// TIA Portal V19 export
DATA_BLOCK "PnPnLeftX2P1PNPortStatus_DB"   // DB11
// stored: InstanceOfName PN Port Status, InstanceOfType FB
"PN Port Status"
   // VAR_INPUT
   //    HW_ID : HW_IO;
   //    Update : Bool;
   // END_VAR
   // VAR_OUTPUT
   //    Connected : Bool;
   // END_VAR
   // VAR
   //    Updated_ReqP : Bool;
   //    Updated_Req : Bool;
   //    RDREC_Instance { S7_SetPoint := 'True'} : RDREC;
   // END_VAR
BEGIN
END_DATA_BLOCK
